// TIA Portal V20 export
TYPE "IO_Device_Test_Parameters"
   STRUCT
      Reset_PLC_Functional_Test_2 : Bool;
      Reset_PLC_Functional_Test_4 : Bool;
      Reset_PLC_Functional_Test_6 : Bool;
      Reset_PLC_Functional_Test_8 : Bool;
      Reset_PLC_Functional_Test_10 : Bool;
      Reset_PLC_Functional_Test_12 : Bool;
      Reset_PLC_Functional_Test_14 : Bool;
      Reset_PLC_Functional_Test_16 : Bool;
      Reset_PLC_Functional_Test_18 : Bool;
      Reset_PLC_Functional_Test_20 : Bool;
      Reset_PLC_Functional_Test_22 : Bool;
      Reset_PLC_Functional_Test_24 : Bool;
      Reset_PLC_Functional_Test_26 : Bool;
      Reset_PLC_Functional_Test_28 : Bool;
      Reset_PLC_Functional_Test_30 : Bool;
      Status : Bool;
      Voltage_Read : UInt;
      Min_Electrical_Current : UInt;
      Max_Electrical_Current : UInt;
      Time_End_Electrical_Current_Test : Time;
      Time_Start_Visual_Test : Time;
   END_STRUCT;
END_TYPE
